FUNCTION_BLOCK SORT (* Template for a Basic Function Block Type *)
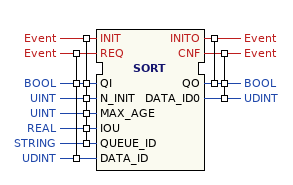
  EVENT_INPUT
    INIT WITH QI, N_INIT, MAX_AGE, IOU, QUEUE_ID; (* Initialization Request *)
    REQ WITH QI, DATA_ID; (* Normal Execution Request *)
  END_EVENT
  EVENT_OUTPUT
    INITO WITH QO; (* Initialization Confirm *)
    CNF WITH QO, DATA_ID0; (* Execution Confirmation *)
  END_EVENT
  VAR_INPUT
    QI : BOOL; (* Input event qualifier *)
    N_INIT : UINT;
    MAX_AGE : UINT;
    IOU : REAL;
    QUEUE_ID : STRING;
    DATA_ID : UDINT;
  END_VAR
  VAR_OUTPUT
    QO : BOOL; (* Output event qualifier *)
    DATA_ID0 : UDINT;
  END_VAR
END_FUNCTION_BLOCK
